FUNCTION_BLOCK Foo
VAR
    Counter : UINT := 0;
END_VAR

Counter := Counter + 1;

END_FUNCTION_BLOCK

(* stored: Version 1.1.0.1, ProductVersion 3.1.4024.4
   POU Foo: Id {d933c360-a8c5-4fa1-a388-adc180a481d2}, SpecialFunc None *)
